TYPE T_PROCESS : DWORD; END_TYPE

(* stored: Version 1.1.0.1, ProductVersion 3.1.4026.18
   DUT T_PROCESS: Id {c93388e7-e291-41bb-b844-ea869e548cbd} *)
